{attribute 'qualified_only'}
VAR_GLOBAL
		// Endschalter Links
	B1 : BOOL; 
	// Endschalter REchts
	B2: BOOL;
	// Thermorelais
	F1: BOOL;
	// Taster Start
	S1: BOOL;
	// Taster NotHalt
	S2: BOOL;
	// Taster Reset
	S3: BOOL;
END_VAR

(* stored: Version 1.1.0.1, ProductVersion 3.1.4022.7
   GVL AdsInput: Id {c2d05302-d374-4f85-80dd-41006a3e3277} *)
